{attribute 'qualified_only'}
VAR_GLOBAL
	fEncoder1Rad AT %I* : REAL;
	fEncoder2Rad AT %I* : REAL;
	fEncoder3Rad AT %I* : REAL;
	fTelescopeDistance_mm AT %I* : REAL;
	fXRotDeg AT %I* : REAL;
	fYRotDeg AT %I* : REAL;
	bSensorDataLost : BOOL;
END_VAR

(* stored: Version 1.1.0.1, ProductVersion 3.1.4024.12
   GVL G_SensorInput: Id {eaec8836-4265-4e28-b2a0-04d44cc088be} *)
